PROGRAM MAIN

VAR
	
	
	
	aInputs AT %I* : ARRAY[1..8] OF BOOL;
	aOutputs AT %Q* : ARRAY[1..8] OF BOOL;
	
	bGreenBtn    : POINTER TO BOOL:= ADR(aInputs[1]);
	bRedBtn		: POINTER TO BOOL:= ADR(aInputs[2]);
	bLight : POINTER TO BOOL := ADR(aOutputs[1]);
	//bTestRef1 := ADR(aInputs[1]);
	
	//input : fbDigitalInput(ioBitRef := bGreenBtn);
	//input2 : fbDigitalIO(ioBitRef := bTestRef1);
	//fbStartInput : fbDigitalInput(ioBitRef := (aInputs[1]));
	//fbStopInput : fbDigitalInput(ioBitRef := (aInputs[2]));
	//fbLightOutput : fbDigitalOutput(ioBitRef := (aOutputs[1]));
END_VAR




aOutputs[8] := aInputs[8]; // Output 8 mirrors input 8




//bGreenBtn := aInputs[1];



IF bGreenBtn^ THEN
		bLight^:=TRUE;
		//fbLightOutput.Set(TRUE);
ELSE
		bLight^:=FALSE;
		//fbLightOutput.Set(FALSE);	
END_IF

(*
CASE CurrentState OF
    E_MyStates.STATE_IDLE:
        // Actions for the IDLE state
        Output1 := FALSE;
        Output2 := FALSE;

    E_MyStates.STATE_RUNNING:
        // Actions for the RUNNING state
        Output1 := TRUE;
        Output2 := TRUE;

    E_MyStates.STATE_STOPPED:
        // Actions for the STOPPED state
        Output1 := FALSE;
        Output2 := TRUE;

    E_MyStates.STATE_ERROR:
        // Actions for the ERROR state
        Output1 := TRUE;
        Output2 := FALSE;

ELSE
    // Default actions if CurrentState does not match any defined case
    // This is optional but good practice for handling unexpected values
    Output1 := FALSE;
    Output2 := FALSE;
END_CASE

*)

END_PROGRAM

(* stored: Version 1.1.0.1, ProductVersion 3.1.4024.15
   POU MAIN: Id {2619c018-a97e-4e98-bfde-76b022b13f51}, SpecialFunc None *)
